// TIA Portal V18 export
VAR_GLOBAL   // PLC tag table "Default tag table"
   TestByte AT %MB2500 : Byte;
   RotaryRPMHMI AT %MD534 : Real;   // It is a absolute value, to display on HMI gauge
   PSIcheck AT %MD544 : Real;
   RotaryStopped AT %M568.0 : Bool;
   MUTorqSetKFtLbs AT %MD570 : Real;
   DrillTorqSetKFtLbs AT %MD574 : Real;
END_VAR
VAR_GLOBAL CONSTANT   // user constants
   RigNumber : Real := 0.0;
   "Program Version" : Real := 0.0;
   RotaryEncInvDir : Bool := 0;   // Used to invert the counting of the rotary encoder
END_VAR
